PROGRAM prgPersistent
VAR
	fbUSV		: FB_WritePersistentData_CX81xx;
END_VAR

fbUSV(
	eSaveModeData:= eUSVSaveMode.eSaveWhenPowerfail, 
	bLoadPersistentDataOk=> , 
	bPowerFailDetect=> , 
	bError=> , 
	bySaveProcess=> , 
	dwStorageLast24h=> , 
	udiErrorCode=> );
	
prg_SystemTime();

END_PROGRAM

(* stored: Version 1.1.0.1, ProductVersion 3.1.4024.11
   POU prgPersistent: Id {cf2e0bad-677f-4823-a2bf-489f86d455a8}, SpecialFunc None *)
